// TIA Portal V15.1 export
// export: Created 2020-06-12T07:35:46.6318359Z, ExportSetting None, DisplayName Totally Integrated Automation Portal, DisplayVersion V15.1, DisplayName TIA Portal Openness, DisplayVersion V15.1, DisplayName STEP 7 Professional, DisplayVersion V15.1, DisplayName STEP 7 Safety, DisplayVersion V15.1, DisplayName WinCC Advanced, DisplayVersion V15.1
FUNCTION "ELC_move" : Void   // FC701, FBD
TITLE = Elcectrode Movement Control
{ S7_Optimized_Access := 'TRUE' }
// #_contr_up
// #_contr_dwn
// stored: AutoNumber false, SetENOAutomatically False
   VAR_TEMP
      _GD01_up : Bool;
      _GD01_dwn : Bool;
      _contr_up : Bool;
      _GD01_fst : Bool;
      _GD02_up : Bool;
      _GD02_dwn : Bool;
      _GD02_fst : Bool;
      _GT07_td_req : Bool;
      _contr_dwn : Bool;
      _csf : Bool;
      _man : Bool;
      _fl_auto_up : Bool;
      _fl_td_btn : Bool;
      _set_zero : Bool;
      _LE4M01_auto_on : Bool;
      _td_pos_fst : Real;
      tElcEndPos : Real;
      _td_res_wt : Real;
      tTouchDownLock : Bool;
      tEnFastMoveUp : Bool;
      tEnFastMoveDown : Bool;
      tFastMovePath : Real;
      tCorrectionDelta : Real;
      tSpdIsZero : Bool;
      tSpdIsZero2 : Bool;
      tSpdZero : Real;
      tSpdIsPos : Bool;
      tSpdIsNeg : Bool;
      tLckByMinWgt : Bool;
   END_VAR
   VAR_TEMP   // added for the SCL form of the ladder/FBD networks
      _w1 : Bool;
      _w2 : Bool;
   END_VAR
BEGIN

REGION Network 1: Electrode carriage: power supply
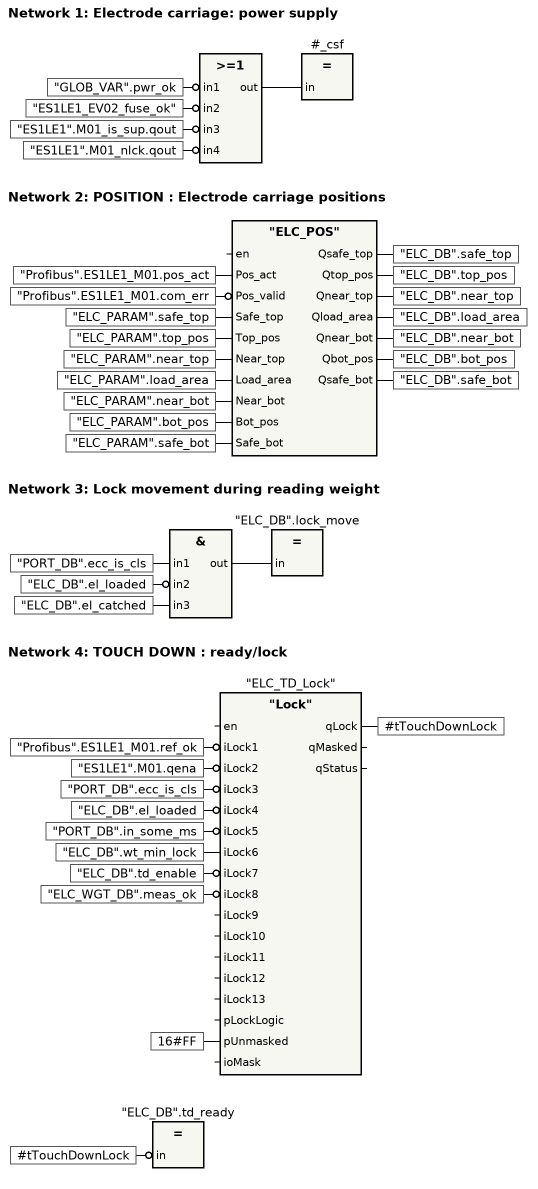
   #_csf := NOT "GLOB_VAR".pwr_ok OR NOT "ES1LE1_EV02_fuse_ok" OR NOT "ES1LE1".M01_is_sup.qout OR NOT "ES1LE1".M01_nlck.qout;
END_REGION

REGION Network 2: POSITION : Electrode carriage positions
   // ECR stroke = 2560 mm
   // ECR Current pipe length = 5650 mm
   // ECR mechanical top position = 6000 mm
   // ECR safe top position = 5980 mm
   "ELC_POS"(Pos_act := "Profibus".ES1LE1_M01.pos_act,
             Pos_valid := NOT "Profibus".ES1LE1_M01.com_err,
             Safe_top := "ELC_PARAM".safe_top,
             Top_pos := "ELC_PARAM".top_pos,
             Near_top := "ELC_PARAM".near_top,
             Load_area := "ELC_PARAM".load_area,
             Near_bot := "ELC_PARAM".near_bot,
             Bot_pos := "ELC_PARAM".bot_pos,
             Safe_bot := "ELC_PARAM".safe_bot,
             Qsafe_top => "ELC_DB".safe_top,
             Qtop_pos => "ELC_DB".top_pos,
             Qnear_top => "ELC_DB".near_top,
             Qload_area => "ELC_DB".load_area,
             Qnear_bot => "ELC_DB".near_bot,
             Qbot_pos => "ELC_DB".bot_pos,
             Qsafe_bot => "ELC_DB".safe_bot);
END_REGION

REGION Network 3: Lock movement during reading weight
   "ELC_DB".lock_move := "PORT_DB".ecc_is_cls AND NOT "ELC_DB".el_loaded AND "ELC_DB".el_catched;
END_REGION

REGION Network 4: TOUCH DOWN : ready/lock
   "ELC_TD_Lock"(iLock1 := NOT "Profibus".ES1LE1_M01.ref_ok,   // "Lock"
                 iLock2 := NOT "ES1LE1".M01.qena,
                 iLock3 := NOT "PORT_DB".ecc_is_cls,
                 iLock4 := NOT "ELC_DB".el_loaded,
                 iLock5 := NOT "PORT_DB".in_some_ms,
                 iLock6 := "ELC_DB".wt_min_lock,
                 iLock7 := NOT "ELC_DB".td_enable,
                 iLock8 := NOT "ELC_WGT_DB".meas_ok,
                 pUnmasked := 16#FF,
                 qLock => #tTouchDownLock);
   "ELC_DB".td_ready := NOT #tTouchDownLock;
END_REGION

REGION Network 5: TOUCH DOWN : finished
   // "MELT_VAR_DB".meas_el_WT_brutto_act
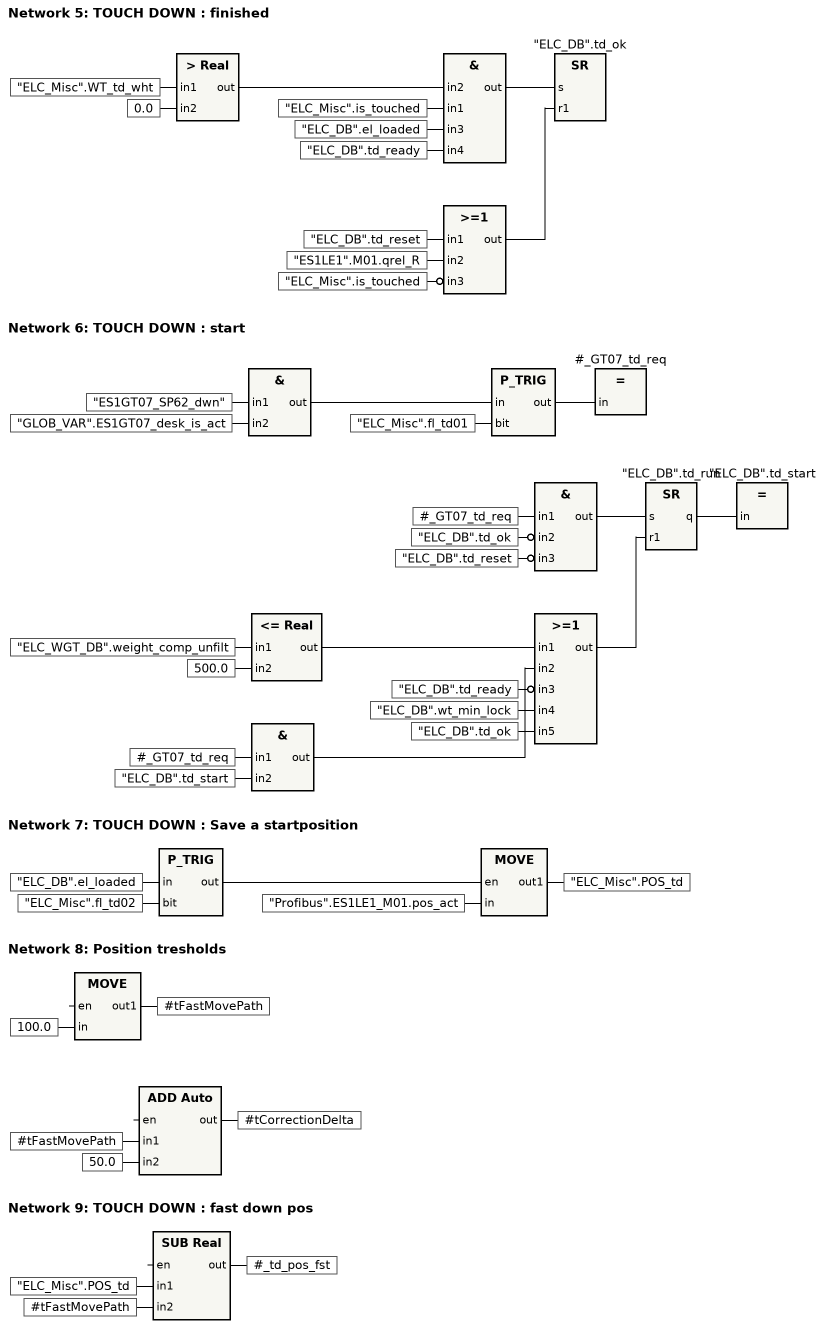
   IF ("ELC_Misc".WT_td_wht > 0.0) AND "ELC_Misc".is_touched AND "ELC_DB".el_loaded AND "ELC_DB".td_ready THEN
       "ELC_DB".td_ok := TRUE;   // SR flip-flop
   END_IF;
   IF "ELC_DB".td_reset OR "ES1LE1".M01.qrel_R OR NOT "ELC_Misc".is_touched THEN
       "ELC_DB".td_ok := FALSE;
   END_IF;
END_REGION

REGION Network 6: TOUCH DOWN : start
   // PuM/2018-05-28: I remove the signal RESET by "GLOB_VAR".ES1GD02_desk_is_act beacuse the TouchDown can be done without desk
   #_w1 := "ES1GT07_SP62_dwn" AND "GLOB_VAR".ES1GT07_desk_is_act;
   #_w2 := #_w1 AND NOT "ELC_Misc".fl_td01;   // rising edge
   "ELC_Misc".fl_td01 := #_w1;
   #_GT07_td_req := #_w2;
   IF #_GT07_td_req AND NOT "ELC_DB".td_ok AND NOT "ELC_DB".td_reset THEN
       "ELC_DB".td_run := TRUE;   // SR flip-flop
   END_IF;
   IF ("ELC_WGT_DB".weight_comp_unfilt <= 500.0) OR (#_GT07_td_req AND "ELC_DB".td_start) OR NOT "ELC_DB".td_ready OR "ELC_DB".wt_min_lock OR "ELC_DB".td_ok THEN
       "ELC_DB".td_run := FALSE;
   END_IF;
   "ELC_DB".td_start := "ELC_DB".td_run;
END_REGION

REGION Network 7: TOUCH DOWN : Save a startposition
   #_w1 := "ELC_DB".el_loaded AND NOT "ELC_Misc".fl_td02;   // rising edge
   "ELC_Misc".fl_td02 := "ELC_DB".el_loaded;
   IF #_w1 THEN "ELC_Misc".POS_td := "Profibus".ES1LE1_M01.pos_act; END_IF;
END_REGION

REGION Network 8: Position tresholds
   #tFastMovePath := 100.0;
   #tCorrectionDelta := #tFastMovePath + 50.0;
END_REGION

REGION Network 9: TOUCH DOWN : fast down pos
   #_td_pos_fst := "ELC_Misc".POS_td - #tFastMovePath;
END_REGION

REGION Network 10: TOUCH DOWN : Correction of the startposition
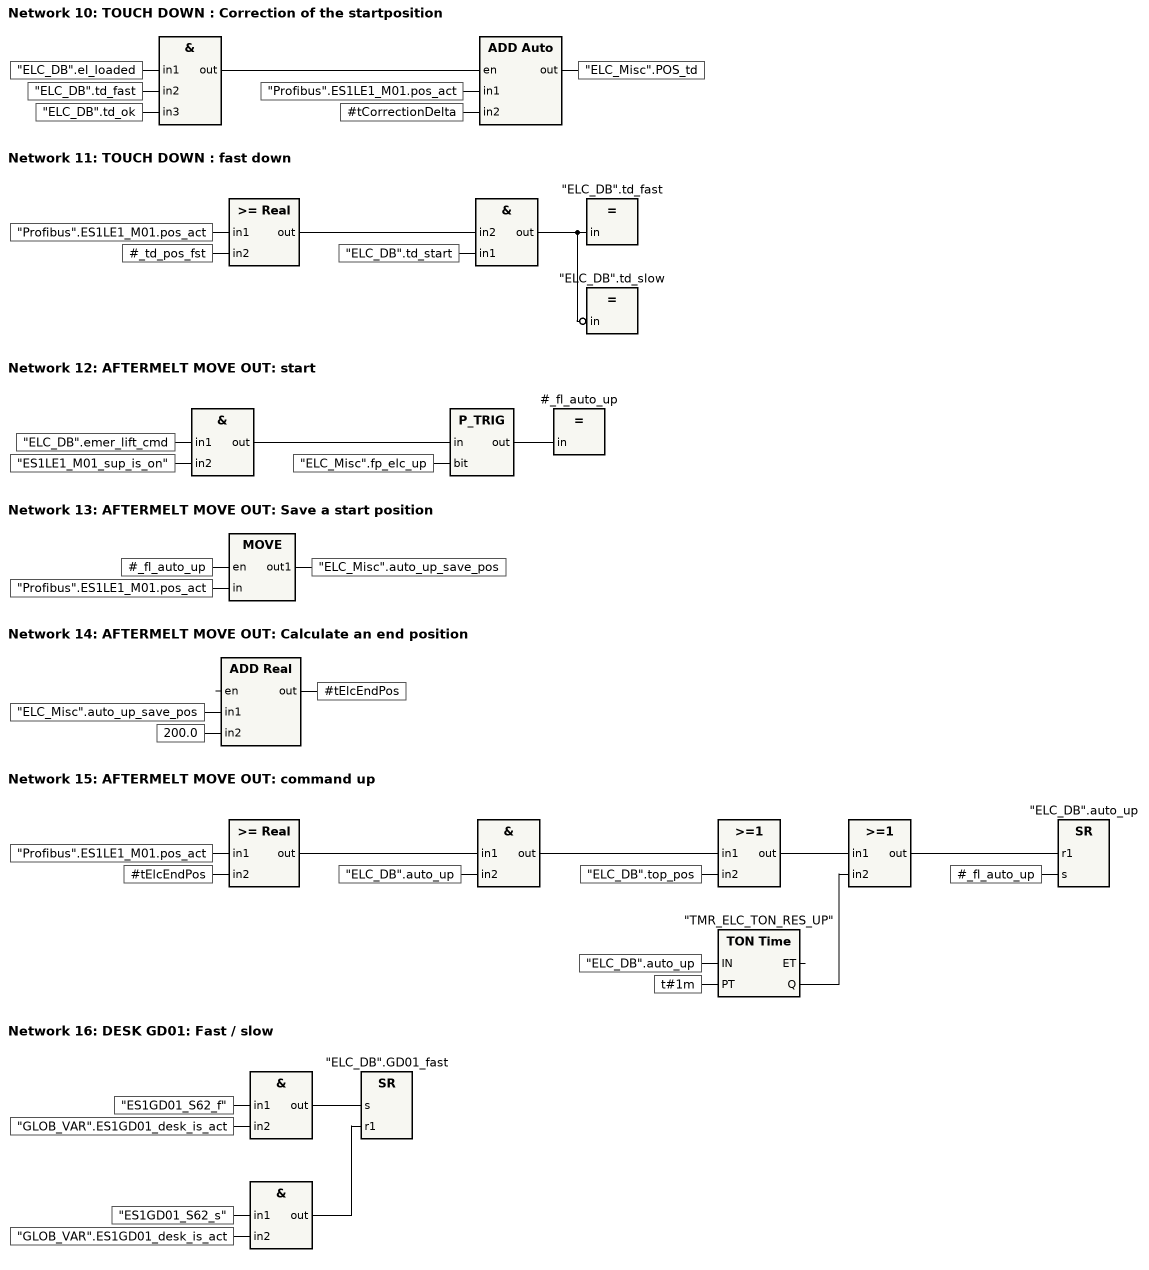
   IF "ELC_DB".el_loaded AND "ELC_DB".td_fast AND "ELC_DB".td_ok THEN
       "ELC_Misc".POS_td := "Profibus".ES1LE1_M01.pos_act + #tCorrectionDelta;
   END_IF;
END_REGION

REGION Network 11: TOUCH DOWN : fast down
   "ELC_DB".td_fast := ("Profibus".ES1LE1_M01.pos_act >= #_td_pos_fst) AND "ELC_DB".td_start;
   "ELC_DB".td_slow := NOT "ELC_DB".td_fast;
END_REGION

REGION Network 12: AFTERMELT MOVE OUT: start
   #_w1 := "ELC_DB".emer_lift_cmd AND "ES1LE1_M01_sup_is_on";
   #_w2 := #_w1 AND NOT "ELC_Misc".fp_elc_up;   // rising edge
   "ELC_Misc".fp_elc_up := #_w1;
   #_fl_auto_up := #_w2;
END_REGION

REGION Network 13: AFTERMELT MOVE OUT: Save a start position
   IF #_fl_auto_up THEN "ELC_Misc".auto_up_save_pos := "Profibus".ES1LE1_M01.pos_act; END_IF;
END_REGION

REGION Network 14: AFTERMELT MOVE OUT: Calculate an end position
   #tElcEndPos := "ELC_Misc".auto_up_save_pos + 200.0;
END_REGION

REGION Network 15: AFTERMELT MOVE OUT: command up
   "TMR_ELC_TON_RES_UP".TON(IN := "ELC_DB".auto_up, PT := t#1m);
   #_w1 := (("Profibus".ES1LE1_M01.pos_act >= #tElcEndPos) AND "ELC_DB".auto_up) OR "ELC_DB".top_pos OR "TMR_ELC_TON_RES_UP".Q;
   IF #_fl_auto_up THEN
       "ELC_DB".auto_up := TRUE;   // SR flip-flop
   END_IF;
   IF #_w1 THEN "ELC_DB".auto_up := FALSE; END_IF;
END_REGION

REGION Network 16: DESK GD01: Fast / slow
   IF "ES1GD01_S62_f" AND "GLOB_VAR".ES1GD01_desk_is_act THEN
       "ELC_DB".GD01_fast := TRUE;   // SR flip-flop
   END_IF;
   IF "ES1GD01_S62_s" AND "GLOB_VAR".ES1GD01_desk_is_act THEN "ELC_DB".GD01_fast := FALSE; END_IF;
END_REGION

REGION Network 17: DESK GD01: commands
   // PuM: why there are not external stops?
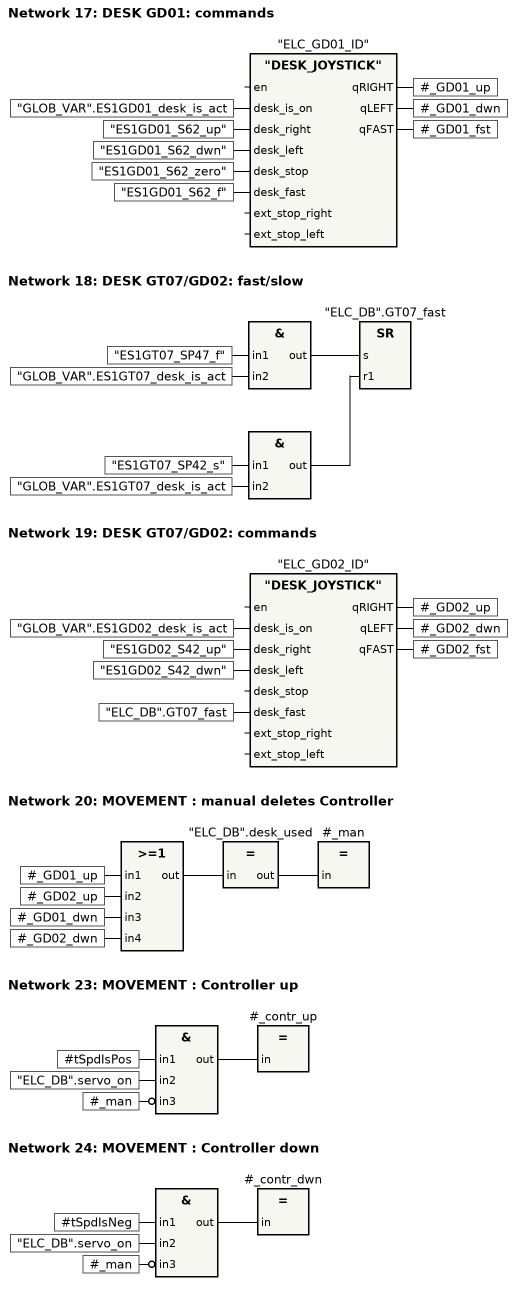
   "ELC_GD01_ID"(desk_is_on := "GLOB_VAR".ES1GD01_desk_is_act,   // "DESK_JOYSTICK"
                 desk_right := "ES1GD01_S62_up",
                 desk_left := "ES1GD01_S62_dwn",
                 desk_stop := "ES1GD01_S62_zero",
                 desk_fast := "ES1GD01_S62_f",
                 qRIGHT => #_GD01_up,
                 qLEFT => #_GD01_dwn,
                 qFAST => #_GD01_fst);
END_REGION

REGION Network 18: DESK GT07/GD02: fast/slow
   IF "ES1GT07_SP47_f" AND "GLOB_VAR".ES1GT07_desk_is_act THEN
       "ELC_DB".GT07_fast := TRUE;   // SR flip-flop
   END_IF;
   IF "ES1GT07_SP42_s" AND "GLOB_VAR".ES1GT07_desk_is_act THEN "ELC_DB".GT07_fast := FALSE; END_IF;
END_REGION

REGION Network 19: DESK GT07/GD02: commands
   "ELC_GD02_ID"(desk_is_on := "GLOB_VAR".ES1GD02_desk_is_act,   // "DESK_JOYSTICK"
                 desk_right := "ES1GD02_S42_up",
                 desk_left := "ES1GD02_S42_dwn",
                 desk_fast := "ELC_DB".GT07_fast,
                 qRIGHT => #_GD02_up,
                 qLEFT => #_GD02_dwn,
                 qFAST => #_GD02_fst);
END_REGION

REGION Network 20: MOVEMENT : manual deletes Controller
   "ELC_DB".desk_used := #_GD01_up OR #_GD02_up OR #_GD01_dwn OR #_GD02_dwn;
   #_man := "ELC_DB".desk_used;
END_REGION

REGION Network 21 (SCL): MOVEMENT : direction recognition
   // NOTE: The Lenze servo drive accepts the setpoint above 0.1 mm/min (for a start, but can keep after start)
   #tSpdZero := 0.05;
   #tSpdIsPos := "ELC_DB".servo_set > #tSpdZero;
   #tSpdIsNeg := "ELC_DB".servo_set < -#tSpdZero;
END_REGION

REGION Network 22 (SCL): MOVEMENT : speed setpoint monitoring
   // NOTE: The Lenze servo drive accepts the setpoint above 0.1 mm/min (for a start, but can keep after start)
   #tSpdIsZero := NOT #tSpdIsPos AND NOT #tSpdIsNeg;
   #tSpdIsZero2 := ABS("ELC_DB".servo_set) <= 4 * #tSpdZero;
END_REGION

REGION Network 23: MOVEMENT : Controller up
   #_contr_up := #tSpdIsPos AND "ELC_DB".servo_on AND NOT #_man;
END_REGION

REGION Network 24: MOVEMENT : Controller down
   #_contr_dwn := #tSpdIsNeg AND "ELC_DB".servo_on AND NOT #_man;
END_REGION

REGION Network 25: MOVEMENT : disable runtime errors
   // To avoid the errors generation within servo mode by zero speed
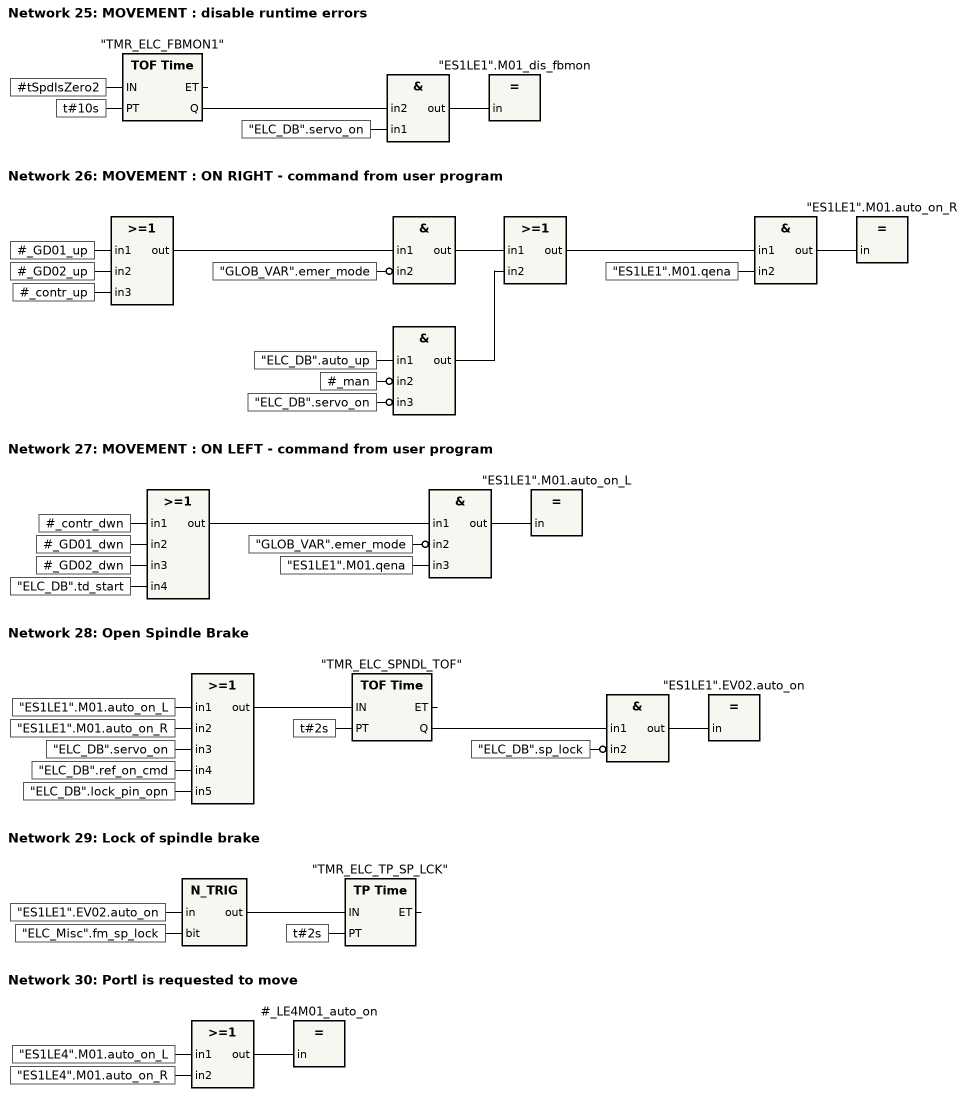
   "TMR_ELC_FBMON1".TOF(IN := #tSpdIsZero2, PT := t#10s);
   "ES1LE1".M01_dis_fbmon := "TMR_ELC_FBMON1".Q AND "ELC_DB".servo_on;
END_REGION

REGION Network 26: MOVEMENT : ON RIGHT - command from user program
   "ES1LE1".M01.auto_on_R := (((#_GD01_up OR #_GD02_up OR #_contr_up) AND NOT "GLOB_VAR".emer_mode) OR ("ELC_DB".auto_up AND NOT #_man AND NOT "ELC_DB".servo_on)) AND "ES1LE1".M01.qena;
END_REGION

REGION Network 27: MOVEMENT : ON LEFT - command from user program
   "ES1LE1".M01.auto_on_L := (#_contr_dwn OR #_GD01_dwn OR #_GD02_dwn OR "ELC_DB".td_start) AND NOT "GLOB_VAR".emer_mode AND "ES1LE1".M01.qena;
END_REGION

REGION Network 28: Open Spindle Brake
   "TMR_ELC_SPNDL_TOF".TOF(IN := "ES1LE1".M01.auto_on_L OR "ES1LE1".M01.auto_on_R OR "ELC_DB".servo_on OR "ELC_DB".ref_on_cmd OR "ELC_DB".lock_pin_opn,
                           PT := t#2s);
   "ES1LE1".EV02.auto_on := "TMR_ELC_SPNDL_TOF".Q AND NOT "ELC_DB".sp_lock;
END_REGION

REGION Network 29: Lock of spindle brake
   #_w1 := NOT "ES1LE1".EV02.auto_on AND "ELC_Misc".fm_sp_lock;   // falling edge
   "ELC_Misc".fm_sp_lock := "ES1LE1".EV02.auto_on;
   "TMR_ELC_TP_SP_LCK".TP(IN := #_w1, PT := t#2s);
END_REGION

REGION Network 30: Portl is requested to move
   #_LE4M01_auto_on := "ES1LE4".M01.auto_on_L OR "ES1LE4".M01.auto_on_R;
END_REGION

REGION Network 31: MOVEMENT : LOCK up
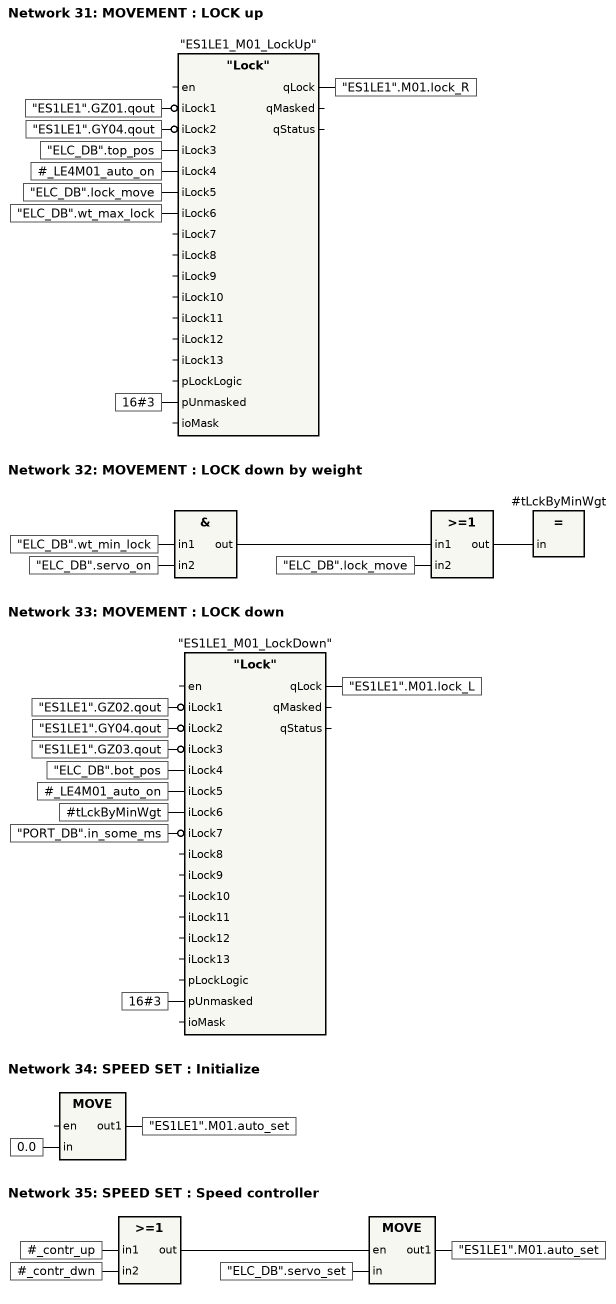
   "ES1LE1_M01_LockUp"(iLock1 := NOT "ES1LE1".GZ01.qout,   // "Lock"
                       iLock2 := NOT "ES1LE1".GY04.qout,
                       iLock3 := "ELC_DB".top_pos,
                       iLock4 := #_LE4M01_auto_on,
                       iLock5 := "ELC_DB".lock_move,
                       iLock6 := "ELC_DB".wt_max_lock,
                       pUnmasked := 16#3,
                       qLock => "ES1LE1".M01.lock_R);
END_REGION

REGION Network 32: MOVEMENT : LOCK down by weight
   #tLckByMinWgt := ("ELC_DB".wt_min_lock AND "ELC_DB".servo_on) OR "ELC_DB".lock_move;
END_REGION

REGION Network 33: MOVEMENT : LOCK down
   "ES1LE1_M01_LockDown"(iLock1 := NOT "ES1LE1".GZ02.qout,   // "Lock"
                         iLock2 := NOT "ES1LE1".GY04.qout,
                         iLock3 := NOT "ES1LE1".GZ03.qout,
                         iLock4 := "ELC_DB".bot_pos,
                         iLock5 := #_LE4M01_auto_on,
                         iLock6 := #tLckByMinWgt,
                         iLock7 := NOT "PORT_DB".in_some_ms,
                         pUnmasked := 16#3,
                         qLock => "ES1LE1".M01.lock_L);
END_REGION

REGION Network 34: SPEED SET : Initialize
   "ES1LE1".M01.auto_set := 0.0;
END_REGION

REGION Network 35: SPEED SET : Speed controller
   IF #_contr_up OR #_contr_dwn THEN "ES1LE1".M01.auto_set := "ELC_DB".servo_set; END_IF;
END_REGION

REGION Network 36: SPEED SET : Touch-down
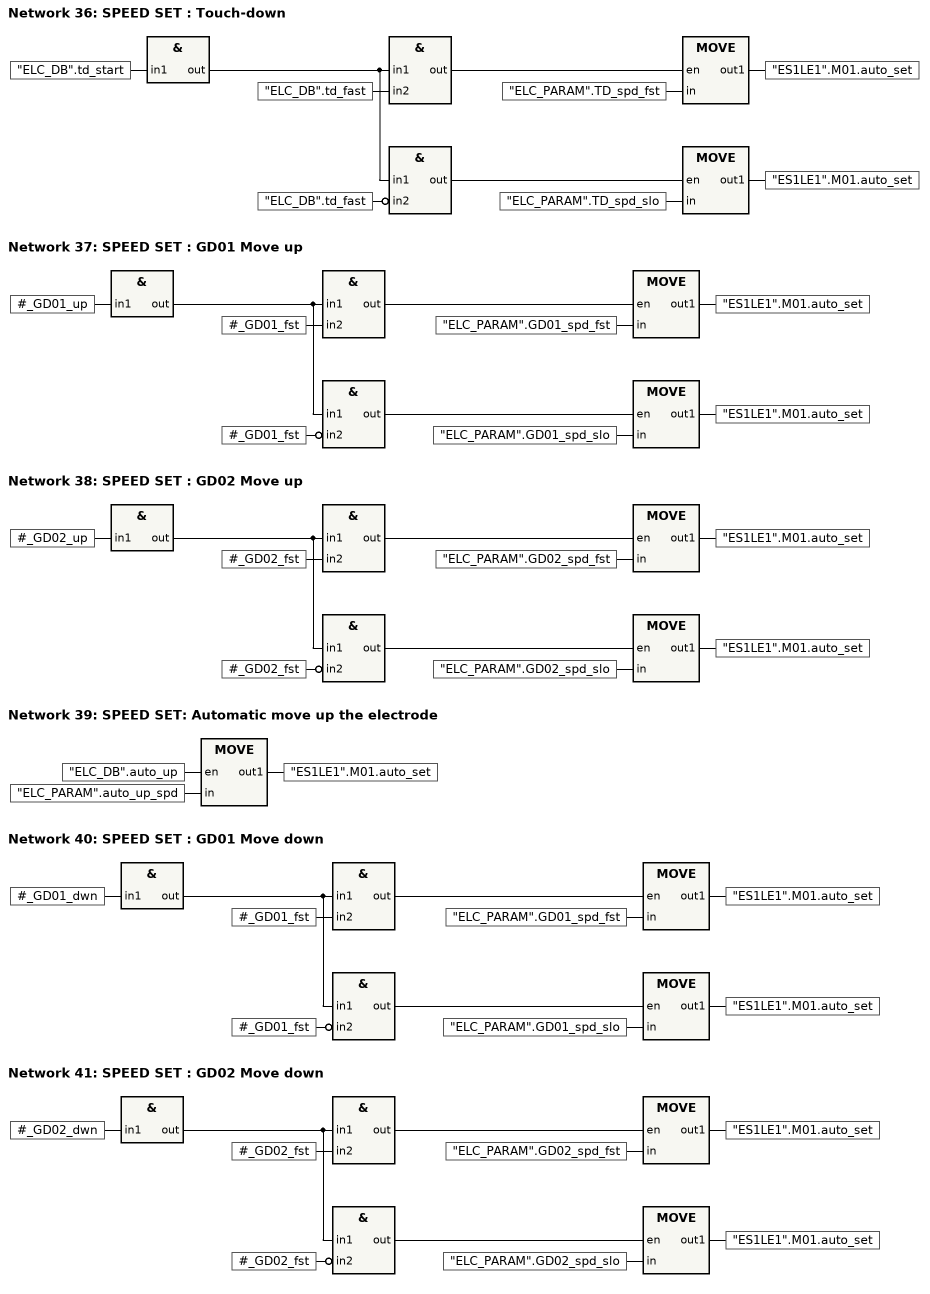
   IF "ELC_DB".td_start AND "ELC_DB".td_fast THEN "ES1LE1".M01.auto_set := "ELC_PARAM".TD_spd_fst; END_IF;
   IF "ELC_DB".td_start AND NOT "ELC_DB".td_fast THEN
       "ES1LE1".M01.auto_set := "ELC_PARAM".TD_spd_slo;
   END_IF;
END_REGION

REGION Network 37: SPEED SET : GD01 Move up
   // "ESM_ELC_DAT_GEN".td_fast
   // #_GD02_up
   IF #_GD01_up AND #_GD01_fst THEN "ES1LE1".M01.auto_set := "ELC_PARAM".GD01_spd_fst; END_IF;
   IF #_GD01_up AND NOT #_GD01_fst THEN "ES1LE1".M01.auto_set := "ELC_PARAM".GD01_spd_slo; END_IF;
END_REGION

REGION Network 38: SPEED SET : GD02 Move up
   // "ESM_ELC_DAT_GEN".td_fast
   // #_GD02_up
   IF #_GD02_up AND #_GD02_fst THEN "ES1LE1".M01.auto_set := "ELC_PARAM".GD02_spd_fst; END_IF;
   IF #_GD02_up AND NOT #_GD02_fst THEN "ES1LE1".M01.auto_set := "ELC_PARAM".GD02_spd_slo; END_IF;
END_REGION

REGION Network 39: SPEED SET: Automatic move up the electrode
   IF "ELC_DB".auto_up THEN "ES1LE1".M01.auto_set := "ELC_PARAM".auto_up_spd; END_IF;
END_REGION

REGION Network 40: SPEED SET : GD01 Move down
   IF #_GD01_dwn AND #_GD01_fst THEN "ES1LE1".M01.auto_set := "ELC_PARAM".GD01_spd_fst; END_IF;
   IF #_GD01_dwn AND NOT #_GD01_fst THEN "ES1LE1".M01.auto_set := "ELC_PARAM".GD01_spd_slo; END_IF;
END_REGION

REGION Network 41: SPEED SET : GD02 Move down
   IF #_GD02_dwn AND #_GD02_fst THEN "ES1LE1".M01.auto_set := "ELC_PARAM".GD02_spd_fst; END_IF;
   IF #_GD02_dwn AND NOT #_GD02_fst THEN "ES1LE1".M01.auto_set := "ELC_PARAM".GD02_spd_slo; END_IF;
END_REGION

REGION Network 43: SPEED SET : Enable the fast up movement
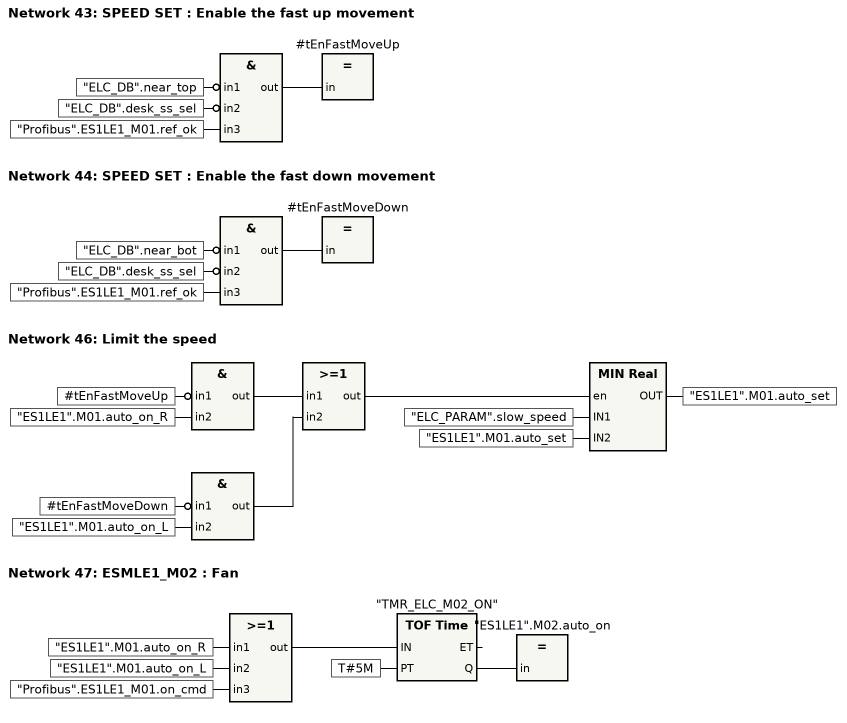
   #tEnFastMoveUp := NOT "ELC_DB".near_top AND NOT "ELC_DB".desk_ss_sel AND "Profibus".ES1LE1_M01.ref_ok;
END_REGION

REGION Network 44: SPEED SET : Enable the fast down movement
   #tEnFastMoveDown := NOT "ELC_DB".near_bot AND NOT "ELC_DB".desk_ss_sel AND "Profibus".ES1LE1_M01.ref_ok;
END_REGION

REGION Network 45 (SCL): Limit of speed
   "ES1LE1".M01.auto_set := LIMIT_REAL(MN := - "ELC_PARAM".fast_speed
                                       , IN := "ES1LE1".M01.auto_set
                                       , MX := "ELC_PARAM".fast_speed);
END_REGION

REGION Network 46: Limit the speed
   IF (NOT #tEnFastMoveUp AND "ES1LE1".M01.auto_on_R) OR (NOT #tEnFastMoveDown AND "ES1LE1".M01.auto_on_L) THEN
       "ES1LE1".M01.auto_set := MIN(IN1 := "ELC_PARAM".slow_speed, IN2 := "ES1LE1".M01.auto_set);
   END_IF;
END_REGION

REGION Network 47: ESMLE1_M02 : Fan
   "TMR_ELC_M02_ON".TOF(IN := "ES1LE1".M01.auto_on_R OR "ES1LE1".M01.auto_on_L OR "Profibus".ES1LE1_M01.on_cmd,
                        PT := T#5M);
   "ES1LE1".M02.auto_on := "TMR_ELC_M02_ON".Q;
END_REGION
END_FUNCTION
